// TwinCAT 3 PLC project PLC_Project
// ProgramVersion: 3.1.4023.0
// libraries:
//   Tc2_SerialCom, * (Beckhoff Automation GmbH)
//   Tc2_Standard, * (Beckhoff Automation GmbH)
//   Tc2_System, * (Beckhoff Automation GmbH)
//   Tc2_Utilities, * (Beckhoff Automation GmbH)
//   Tc3_Module, * (Beckhoff Automation GmbH)
// project tree:
//   DUTs/ ActivationStatus.TcDUT, GCControllerMode.TcDUT (not stored), GuidanceSystemSTM.TcDUT (not stored), HighLevelCondition.TcDUT (not stored), LEDColor.TcDUT, LEDMode.TcDUT (not stored), LevitationSystemSTM.TcDUT (not stored), OperationControlCommands.TcDUT (not stored), ServiceModuleSTM.TcDUT (not stored), SubLevelCondition.TcDUT (not stored), TGControllerMode.TcDUT, TopLevelSTM.TcDUT, XMCCommands.TcDUT (not stored)
//   OOPs/ FB_HighLevelSystem.TcPOU (not stored), ITF_HighLevelSystem.TcIO (not stored), ITF_SubSystem.TcIO (not stored)
//   / PlcTask.TcTTO
//   POUs/AccelerationSensor/ AccelerationSensor.TcGVL, FB_SerialComRS232.TcPOU (not stored)
//   POUs/BoxLED/ BoxLED.TcGVL
//   POUs/DistanceSensor/ DistanceSensor.TcGVL (not stored), FB_SerialComRS422.TcPOU (not stored)
//   POUs/ FB_AccelerationSensor.TcPOU, FB_BoxLED.TcPOU, FB_DistanceSensor.TcPOU, FB_RGBLED.TcPOU, FB_Test.TcPOU, MAIN.TcPOU, TEST.TcPOU
//   POUs/RGBLED/ RGBLED.TcGVL (not stored)
// real-time tasks:
//   TASK PlcTask: cycle T#1ms, priority 20, ADS port 350
// I/O:
//   DEVICE Gerät 1 (EtherCAT), AmsNetId 10.183.66.136.2.1
//     Klemme 1 (EK1100) [EK1100 EtherCAT-Koppler (2A E-Bus)]
//       Klemme 2 (EL6021) [EL6021 Schnittstelle (RS422/485)]
//       Klemme 3 (EL6001) [EL6001 Schnittstelle (RS232)]
//       Klemme 4 (EL6001) [EL6001 Schnittstelle (RS232)]
//       Klemme 5 (EL2564) [EL2564 4 K. LED-Ausgang, 5...48 V DC, 4 A, RGBW]
//       Klemme 7 (EL9011) [EL9011 Endklemme]
//     Box 6 (CX2040 EtherCAT slave) [CX2040 EtherCAT slave]
// variable links:
//   PLC Project/PLC Project Instance <-> Device 1 (EtherCAT)/Term 1 (EK1100)/Term 3 (EL6001)
//     PlcTask Inputs/AccelerationSensor.stEL6001InIMU1 @bit {16..184 step 8} <-> COM Inputs/Data In {0..21}  (22 links)
//     PlcTask Inputs/AccelerationSensor.stEL6001InIMU1 <-> COM Inputs/Status
//     PlcTask Outputs/AccelerationSensor.stEL6001OutIMU1 <-> COM Outputs/Ctrl
//     PlcTask Outputs/AccelerationSensor.stEL6001OutIMU1 @bit {16..184 step 8} <-> COM Outputs/Data Out {0..21}  (22 links)
//   PLC Project/PLC Project Instance <-> Device 1 (EtherCAT)/Term 1 (EK1100)/Term 4 (EL6001)
//     PlcTask Inputs/AccelerationSensor.stEL6001InIMU2 @bit {16..184 step 8} <-> COM Inputs/Data In {0..21}  (22 links)
//     PlcTask Inputs/AccelerationSensor.stEL6001InIMU2 <-> COM Inputs/Status
//     PlcTask Outputs/AccelerationSensor.stEL6001OutIMU2 <-> COM Outputs/Ctrl
//     PlcTask Outputs/AccelerationSensor.stEL6001OutIMU2 @bit {16..184 step 8} <-> COM Outputs/Data Out {0..21}  (22 links)

CONFIGURATION PLC_Project
    RESOURCE PLC ON TwinCAT3
        TASK PlcTask(INTERVAL := T#1ms, PRIORITY := 20);
        PROGRAM TEST WITH PlcTask : TEST;
    END_RESOURCE
END_CONFIGURATION

// ---- DUTs/ActivationStatus.TcDUT
{attribute 'qualified_only'}
{attribute 'strict'}
TYPE ActivationStatus :
(
	Disabled,
	Enabled
);
END_TYPE

// ---- DUTs/LEDColor.TcDUT
{attribute 'qualified_only'}
{attribute 'strict'}
TYPE LEDColor :
(
	Off,
	Red,
	Green,
	Blue
);
END_TYPE

// ---- DUTs/TGControllerMode.TcDUT
{attribute 'qualified_only'}
{attribute 'strict'}
TYPE TGControllerMode :
(
	IControl,
	PControl
);
END_TYPE

// ---- DUTs/TopLevelSTM.TcDUT
{attribute 'qualified_only'}
{attribute 'strict'}
{attribute 'to_string'}
TYPE TopLevelSTM :
(
	STARTUP,
	READY,
	OPERATIONAL,
	SHUTDOWN,
	ERROR
)USINT;
END_TYPE

// ---- POUs/AccelerationSensor/AccelerationSensor.TcGVL
VAR_GLOBAL
	stEL6001InIMU1 AT %I*	: EL6inData22B;		//**To EL6021 Inputs**
	stEL6001OutIMU1 AT %Q*	: EL6outData22B;	//**To EL6021 Outputs**
	
	stEL6001InIMU2 AT %I*	: EL6inData22B;		//**To EL6021 Inputs**
	stEL6001OutIMU2 AT %Q*	: EL6outData22B;	//**To EL6021 Outputs**
END_VAR

// ---- POUs/BoxLED/BoxLED.TcGVL
{attribute 'qualified_only'}
VAR_GLOBAL
	iWhite AT %Q* : INT;					//**To EL2564 PWM Outputs Channel 4 (PWM output)**
	
	bWhiteError AT %I* : BOOL;				//**To EL2564 PWM Inputs Channel 4 (Status -> Error)**
	bWhiteWarning AT %I* : BOOL;			//**To EL2564 PWM Inputs Channel 4 (Status -> Warning)**
END_VAR

// ---- POUs/TEST.TcPOU
PROGRAM TEST
VAR
	fbTest : FB_Test;
	
	i : INT;
END_VAR

i := fbTest.Prop;

END_PROGRAM

// ---- POUs/FB_Test.TcPOU
FUNCTION_BLOCK FB_Test
VAR_INPUT
END_VAR
VAR_OUTPUT
END_VAR
VAR
	b : BOOL;
END_VAR

PROPERTY PUBLIC Prop : INT
GET
VAR
	counter : UDINT;
END_VAR
IF b THEN
	counter := counter + 1;
END_IF

IF counter = 1000 THEN
	Prop := 999;
END_IF
END_GET
SET
END_SET
END_PROPERTY

END_FUNCTION_BLOCK

// ---- POUs/FB_AccelerationSensor.TcPOU
FUNCTION_BLOCK FB_AccelerationSensor IMPLEMENTS ITF_SubSystem
VAR_IN_OUT
	stRS232Inputs : EL6inData22B;
	stRS232Outputs : EL6outData22B;
END_VAR
VAR_OUTPUT
	aAccelerationValues : ARRAY [0..2] OF REAL;
END_VAR
VAR
	//Local
	fbEL6001	: FB_SerialComRS232;
	
	fPacketRate : REAL := 0;
	bStartPacketCount : BOOL;
	
	fbTimer : TON;
	fbReset : TON;
	fbTrigger : R_TRIG;
	nCounter1 : UDINT;
	nCounter2 : UDINT;
	aPackets : ARRAY [0..9] OF UDINT;
	i : UDINT := 0;
	nSum : UDINT := 0;
	bTrigger : BOOL := FALSE;
	
	//ErrorBits
	bCommunicationError : BIT;
	bOutOfRange : BIT;
END_VAR
VAR CONSTANT
	fGravitationalAcceleration : REAL := 9.81;  					//in m/s^2
END_VAR

fbEL6001(stEL6001In:=stRS232Inputs, stEL6001Out:=stRS232Outputs);

aAccelerationValues := fbEL6001.aAcceleration;

doPacketCount();

METHOD PRIVATE doCheckRange : BOOL
VAR_INPUT
	aValues : ARRAY [0..2] OF REAL;
	fMax : REAL;
END_VAR
IF ABS(aValues[0]) <= fMax AND ABS(aValues[1]) <= fMax AND ABS(aValues[2]) <= fMax THEN
	doCheckRange := TRUE;
ELSE
	doCheckRange := FALSE;
END_IF
END_METHOD

METHOD PRIVATE doPacketCount
VAR_INPUT
END_VAR
fbTimer(IN := bStartPacketCount, PT := T#1S);
fbTrigger(CLK := fbTimer.IN);

IF fbTrigger.Q THEN
	nCounter1 := fbEL6001.nReceiveCounter;
END_IF

IF fbTimer.Q THEN
	nCounter2 := fbEL6001.nReceiveCounter;
	aPackets[i] := nCounter2 - nCounter1;
	nSum := nSum + aPackets[i];
	i := i + 1;
	bTrigger := TRUE;
	bStartPacketCount := FALSE;
END_IF

IF i = 10 THEN
	bTrigger := FALSE;
	fPacketRate := (UDINT_TO_REAL(nSum) / UDINT_TO_REAL(i));
	i := 0;
	nSum := 0;
END_IF

fbReset(IN := bTrigger, PT := T#3S);
IF fbReset.Q THEN
	bStartPacketCount := TRUE;
	bTrigger := FALSE;
END_IF
END_METHOD

PROPERTY PUBLIC eCondition : SubLevelCondition
GET
IF nErrorID <> 0 THEN
	eCondition := SubLevelCondition.ERROR;
ELSE
	eCondition := SubLevelCondition.RUN;
END_IF
END_GET
END_PROPERTY

PROPERTY PUBLIC nErrorID : UDINT
GET
IF fbEL6001.eReceiveErrorID <> COMERROR_NOERROR THEN
	bCommunicationError := TRUE;
ELSE
	bCommunicationError := FALSE;
END_IF

bOutOfRange := NOT doCheckRange(aValues:=aAccelerationValues, fMax:=2*fGravitationalAcceleration);


nErrorID.0 := bCommunicationError;
nErrorID.1 := bOutOfRange;
END_GET
END_PROPERTY

END_FUNCTION_BLOCK

// ---- POUs/FB_BoxLED.TcPOU
FUNCTION_BLOCK FB_BoxLED IMPLEMENTS ITF_SubSystem
VAR_INPUT
	eMode : LEDMode;
END_VAR
VAR
	//Local
	iBoxLED : INT;
	fbFlashingTimer : TON;
	bOn : BOOL;
	
	//ErrorBits
	bTemperatureTooHigh : BIT;
	bNoSupplyVoltage : BIT;
END_VAR
VAR CONSTANT
	iIntensity : INT := 32767;				//Intensity [0..32767]
	rDimFactor : REAL := 0.01;				//Percentage (0..100%)
	tSlowFlashingTime : TIME := T#1S;		
	tFastFlashingTime : TIME := T#100MS;
END_VAR

CASE eMode OF
	LEDMode.Off:
			doTurnOn(iBrightness := 0);
	LEDMode.On:
			doTurnOn(iBrightness := iIntensity);
	LEDMode.Dimmed:
			doDimming(rDimmingFactor:=rDimFactor);
	LEDMode.SlowFlashing:
			doFlashing(FlashingTime:=tSlowFlashingTime);
	LEDMode.FastFlashing:
			doFlashing(FlashingTime:=tFastFlashingTime);
END_CASE

doSetClampValues();
doGetClampValues();

METHOD PRIVATE doDimming
VAR_INPUT
	rDimmingFactor : REAL;
END_VAR
iBoxLED := REAL_TO_INT(rDimmingFactor * iIntensity);
END_METHOD

METHOD PRIVATE doFlashing
VAR_INPUT
	FlashingTime : TIME;
END_VAR
fbFlashingTimer(IN:=TRUE, PT:=FlashingTime);
IF fbFlashingTimer.Q THEN
	fbFlashingTimer(IN:=FALSE);
	bOn := NOT bOn;	
END_IF
IF bOn THEN
	iBoxLED := iIntensity;
ELSE
	iBoxLED := 0;
END_IF
END_METHOD

METHOD PRIVATE doGetClampValues
bTemperatureTooHigh := BoxLED.bWhiteWarning;
bNoSupplyVoltage := BoxLED.bWhiteError;
END_METHOD

METHOD PRIVATE doSetClampValues
BoxLED.iWhite := iBoxLED;
END_METHOD

METHOD PRIVATE doTurnOn
VAR_INPUT
	iBrightness : INT;
END_VAR
iBoxLED := iBrightness;
END_METHOD

PROPERTY eCondition : SubLevelCondition
GET
IF nErrorID <> 0 THEN
	eCondition := SubLevelCondition.ERROR;
ELSE
	eCondition := SubLevelCondition.RUN;
END_IF
END_GET
END_PROPERTY

PROPERTY nErrorID : UDINT
GET
nErrorID.0 := bTemperatureTooHigh;
nErrorID.1 := bNoSupplyVoltage;
END_GET
END_PROPERTY

END_FUNCTION_BLOCK

// ---- POUs/FB_DistanceSensor.TcPOU
FUNCTION_BLOCK FB_DistanceSensor IMPLEMENTS ITF_SubSystem
VAR_OUTPUT
	fDistance 			: LREAL;
END_VAR
VAR
	//Local
	fbEL6021			: FB_SerialComRS422;

	//ErrorBits
	bCommunicationError : BIT;
	bOutOfRange 		: BIT;
END_VAR
VAR CONSTANT
	fSMR 		: LREAL := 50.0;				// Start of Measuring Range
	fEMR 		: LREAL := 150.0;				// End of Measuring Range
END_VAR

fbEL6021(stReceiveData:=DistanceSensor.stEL6021In, stTransmitData:=DistanceSensor.stEL6021Out);

fDistance := fbEL6021.fDistance;

METHOD PRIVATE doCheckRange : BOOL
VAR_INPUT
	fDistanceValue : LREAL;
	fMax : LREAL;
	fMin : LREAL;
END_VAR
IF fDistanceValue < fMin OR fDistanceValue > fMax THEN
	doCheckRange := FALSE;
ELSE
	doCheckRange := TRUE;
END_IF
END_METHOD

PROPERTY eCondition : SubLevelCondition
GET
IF nErrorID <> 0 THEN
	eCondition := SubLevelCondition.ERROR;
ELSE
	eCondition := SubLevelCondition.RUN;
END_IF
END_GET
END_PROPERTY

PROPERTY nErrorID : UDINT
GET
IF fbEL6021.eReceiveErrorID <> COMERROR_NOERROR THEN
	bCommunicationError := TRUE;
ELSE
	bCommunicationError := FALSE;
END_IF

bOutOfRange := NOT doCheckRange(fDistanceValue:= fDistance, fMax:=fEMR, fMin:=fSMR);

nErrorID.0 := bCommunicationError;
nErrorID.1 := bOutOfRange;
END_GET
END_PROPERTY

END_FUNCTION_BLOCK

// ---- POUs/FB_RGBLED.TcPOU
FUNCTION_BLOCK FB_RGBLED IMPLEMENTS ITF_SubSystem
VAR_INPUT
	eColor : LEDColor;
END_VAR
VAR
	//Local
	iRedLED : INT;
	iGreenLED : INT;
	iBlueLED : INT;
	
	//ErrorBits
	bRedTemperatureTooHigh : BIT;
	bRedNoSupplyVoltage : BIT;
	bGreenTemperatureTooHigh : BIT;
	bGreenNoSupplyVoltage : BIT;
	bBlueTemperatureTooHigh : BIT;
	bBlueNoSupplyVoltage : BIT;	
END_VAR
VAR CONSTANT
	iMax : INT := 32767;		//Maximum Intensity (100%)
	iMin : INT := 0;			//Off (0%)
END_VAR

CASE eColor OF
	LEDColor.Off:
		iRedLED := iMin;
		iGreenLED := iMin;
		iBlueLED := iMin;
	LEDColor.Red:
		iRedLED := iMax;
		iGreenLED := iMin;
		iBlueLED := iMin;
	LEDColor.Green:
		iRedLED := iMin;
		iGreenLED := iMax;
		iBlueLED := iMin;
	LEDColor.Blue:
		iRedLED := iMin;
		iGreenLED := iMin;
		iBlueLED := iMax;
END_CASE



doSetClampValues();
doGetClampValues();

METHOD PRIVATE doGetClampValues
VAR_INPUT
END_VAR
bRedTemperatureTooHigh := RGBLED.bRedWarning;
bRedNoSupplyVoltage := RGBLED.bRedError;
bGreenTemperatureTooHigh := RGBLED.bGreenWarning;
bGreenNoSupplyVoltage := RGBLED.bGreenError;
bBlueTemperatureTooHigh := RGBLED.bBlueWarning;
bBlueNoSupplyVoltage := RGBLED.bBlueError;
END_METHOD

METHOD PRIVATE doSetClampValues
RGBLED.iRed := iRedLED;
RGBLED.iGreen := iGreenLED;
RGBLED.iBlue := iBlueLED;
END_METHOD

PROPERTY eCondition : SubLevelCondition
GET
IF nErrorID <> 0 THEN
	eCondition := SubLevelCondition.ERROR;
ELSE
	eCondition := SubLevelCondition.RUN;
END_IF
END_GET
END_PROPERTY

PROPERTY nErrorID : UDINT
GET
nErrorID.0 := bRedTemperatureTooHigh;
nErrorID.1 := bRedNoSupplyVoltage;
nErrorID.2 := bGreenTemperatureTooHigh;
nErrorID.3 := bGreenNoSupplyVoltage;
nErrorID.4 := bBlueTemperatureTooHigh;
nErrorID.5 := bBlueNoSupplyVoltage;
END_GET
END_PROPERTY

END_FUNCTION_BLOCK

// ---- POUs/MAIN.TcPOU
PROGRAM MAIN
VAR
	fbDistanceSensor : FB_DistanceSensor;
	fbIMU1 : FB_AccelerationSensor;
	fbIMU2 : FB_AccelerationSensor;
	fbRGBLED : FB_RGBLED;
	fbBoxLED : FB_BoxLED;
	
	aIMU1 : ARRAY [0..2] OF REAL;
	aIMU2 : ARRAY [0..2] OF REAL;
	fDistance : REAL;
	eColor : LEDColor;
	eMode : LEDMode;
	
END_VAR

fbIMU1(stRS232Inputs:=AccelerationSensor.stEL6001InIMU1, stRS232Outputs:=AccelerationSensor.stEL6001OutIMU1);
fbIMU2(stRS232Inputs:=AccelerationSensor.stEL6001InIMU2, stRS232Outputs := AccelerationSensor.stEL6001OutIMU2);
fbDistanceSensor();
fbBoxLED();
fbRGBLED();

aIMU1 := fbIMU1.aAccelerationValues;
aIMU2 := fbIMU2.aAccelerationValues;
fDistance := LREAL_TO_REAL(fbDistanceSensor.fDistance);
fbBoxLED.eMode := eMode;
fbRGBLED.eColor := eColor;

END_PROGRAM
